INTERFACE I_ModuleConfigurationAdapter EXTENDS __SYSTEM.IQueryInterface

METHOD M_ApplyRuntimeConfig : BOOL
VAR_INPUT
	Slot : UINT;
END_VAR
VAR_IN_OUT CONSTANT
	RuntimeConfig : ST_ModuleRuntimeConfig;
END_VAR
VAR_OUTPUT
	ErrorMessage : STRING(255);
END_VAR
END_METHOD

METHOD M_BindReference : BOOL
VAR_INPUT
	Slot : UINT;
	TargetPort : STRING(80);
	BaseUnit : I_BaseUnit;
END_VAR
VAR_OUTPUT
	ErrorMessage : STRING(255);
END_VAR
END_METHOD

METHOD M_ClearSlot : BOOL
VAR_INPUT
	Slot : UINT;
END_VAR
VAR_OUTPUT
	ErrorMessage : STRING(255);
END_VAR
END_METHOD

METHOD M_IsSlotSupported : BOOL
VAR_INPUT
	Slot : UINT;
END_VAR
END_METHOD

METHOD M_RegisterIo : BOOL
VAR_INPUT
	Slot : UINT;
END_VAR
VAR_IN_OUT
	LinkVariableManager : FB_LinkVariableManager;
END_VAR
VAR_OUTPUT
	ModuleSymbol : STRING(255);
	ErrorMessage : STRING(255);
END_VAR
END_METHOD

METHOD M_ValidateReferences : BOOL
VAR_INPUT
	Slot : UINT;
END_VAR
VAR_OUTPUT
	ErrorMessage : STRING(255);
END_VAR
END_METHOD

END_INTERFACE

(* stored: Version 1.1.0.1, ProductVersion 3.1.4026.18
   Itf I_ModuleConfigurationAdapter: Id {055bce4f-fb38-4c9f-b199-2f3782f87113}
   Method M_ApplyRuntimeConfig: Id {08066e30-8002-45e1-bf31-ea50b3896101}
   Method M_BindReference: Id {633f42e5-d351-4476-a3cd-65a0e153027e}
   Method M_ClearSlot: Id {f7f2334b-9437-4993-b725-e2bbdc75ae40}
   Method M_IsSlotSupported: Id {92540036-d15c-49c1-8b13-2efe61569285}
   Method M_RegisterIo: Id {73830a94-6f8e-4d69-9af6-a4f7c72cc99a}
   Method M_ValidateReferences: Id {abbb786d-1b1a-4189-af7f-8bab1b0650ca} *)
